KUKA KRL data list: program_handler.dat

&ACCESS RV3
&PARAM DISKPATH = KRC:\R1\Program\ROS
DEFDAT program_handler PUBLIC
    ; FOLD Custom enumerations
    GLOBAL CONST INT CYCLE_TIME_COUNT = 3
    GLOBAL ENUM ROS_CycleTime NONE_CYCLE_TIME, RSI_4MS, RSI_12MS
    ; ENDFOLD

    CONST INT INTEGER_MAX = 2147483647
    DECL STATE_T statement_state
    DECL MODUS_T command_mode = #SYNC

    ; FOLD Program handler state variables
    DECL ControlMode selected_control_mode = #INACTIVE
    DECL ROS_CycleTime selected_cycle_time = #RSI_12MS
    ; ENDFOLD
ENDDAT
